Staubli VAL3: load.pgx

public program load(string x_sItem, num& x_nResult)
  local string l_sType
  local string l_sMessage
  local num i
begin
  // load the select trajectory..already loaded
  call getTrajType(l_sType)
  if find(pt:libPath(),saveData:sPathTraj)==-1
    pt:libLoad(saveData:sPathTraj+l_sType)
      delay(0)
    if saveData:bDebug
      ? "loading POINT..."+saveData:sPathTraj+l_sType
    endIf
  endIf
  // use the type...
  if isDefined(pt:tTraj[x_sItem])
    // link the frame and all the points
    call pt:link_all(x_sItem)
    // check if link and defined
    pEditPoint=pt:tTraj[x_sItem]
    pEditPoint.sID=x_sItem
  elseIf x_sItem!=""
    // not FOUND
    call language:message(l_sMessage,-7)
    x_nResult=-1
    popUpMsg(l_sMessage+x_sItem)
  endIf
end
